FUNCTION_BLOCK IO_DI32 (* Cartao TM3DI32K da remota TM3BCEIP: separa as 2 words lidas em 32 bits e publica cada bit por symlink, com depurador *)
  (* Standard: 61499-2 *)
  (* Version 1.0, 10/2/2026, Hidryco, Hidryco, Baseado em TM_DI32/TM_DO32 e DI_TESTE; inclui gate de comunicacao *)
  PACKAGE Hidryco.HidrycoLib;
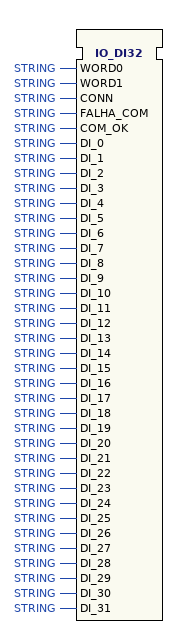
  VAR_INPUT
    WORD0 : STRING; (* Nome do symlink da word 0 do cartao (bits 0-15), ex.: A3_I0_0_15 *)
    WORD1 : STRING; (* Nome do symlink da word 1 do cartao (bits 16-31) *)
    CONN : STRING; (* Nome do symlink connStatusInt da remota, ex.: A2_REMOTA1_CONN_STATUS_INT (obrigatorio: sem ele o cartao fica em falha) *)
    FALHA_COM : STRING; (* Nome do symlink BOOL publicado com a falha de comunicacao do cartao (TRUE = remota offline) *)
    COM_OK : STRING; (* Nome do symlink BOOL publicado com comunicacao OK (TRUE = remota online) *)
    DI_0 : STRING; (* Nome do symlink BOOL publicado para o bit 0 do cartao *)
    DI_1 : STRING; (* Nome do symlink BOOL publicado para o bit 1 do cartao *)
    DI_2 : STRING; (* Nome do symlink BOOL publicado para o bit 2 do cartao *)
    DI_3 : STRING; (* Nome do symlink BOOL publicado para o bit 3 do cartao *)
    DI_4 : STRING; (* Nome do symlink BOOL publicado para o bit 4 do cartao *)
    DI_5 : STRING; (* Nome do symlink BOOL publicado para o bit 5 do cartao *)
    DI_6 : STRING; (* Nome do symlink BOOL publicado para o bit 6 do cartao *)
    DI_7 : STRING; (* Nome do symlink BOOL publicado para o bit 7 do cartao *)
    DI_8 : STRING; (* Nome do symlink BOOL publicado para o bit 8 do cartao *)
    DI_9 : STRING; (* Nome do symlink BOOL publicado para o bit 9 do cartao *)
    DI_10 : STRING; (* Nome do symlink BOOL publicado para o bit 10 do cartao *)
    DI_11 : STRING; (* Nome do symlink BOOL publicado para o bit 11 do cartao *)
    DI_12 : STRING; (* Nome do symlink BOOL publicado para o bit 12 do cartao *)
    DI_13 : STRING; (* Nome do symlink BOOL publicado para o bit 13 do cartao *)
    DI_14 : STRING; (* Nome do symlink BOOL publicado para o bit 14 do cartao *)
    DI_15 : STRING; (* Nome do symlink BOOL publicado para o bit 15 do cartao *)
    DI_16 : STRING; (* Nome do symlink BOOL publicado para o bit 16 do cartao *)
    DI_17 : STRING; (* Nome do symlink BOOL publicado para o bit 17 do cartao *)
    DI_18 : STRING; (* Nome do symlink BOOL publicado para o bit 18 do cartao *)
    DI_19 : STRING; (* Nome do symlink BOOL publicado para o bit 19 do cartao *)
    DI_20 : STRING; (* Nome do symlink BOOL publicado para o bit 20 do cartao *)
    DI_21 : STRING; (* Nome do symlink BOOL publicado para o bit 21 do cartao *)
    DI_22 : STRING; (* Nome do symlink BOOL publicado para o bit 22 do cartao *)
    DI_23 : STRING; (* Nome do symlink BOOL publicado para o bit 23 do cartao *)
    DI_24 : STRING; (* Nome do symlink BOOL publicado para o bit 24 do cartao *)
    DI_25 : STRING; (* Nome do symlink BOOL publicado para o bit 25 do cartao *)
    DI_26 : STRING; (* Nome do symlink BOOL publicado para o bit 26 do cartao *)
    DI_27 : STRING; (* Nome do symlink BOOL publicado para o bit 27 do cartao *)
    DI_28 : STRING; (* Nome do symlink BOOL publicado para o bit 28 do cartao *)
    DI_29 : STRING; (* Nome do symlink BOOL publicado para o bit 29 do cartao *)
    DI_30 : STRING; (* Nome do symlink BOOL publicado para o bit 30 do cartao *)
    DI_31 : STRING; (* Nome do symlink BOOL publicado para o bit 31 do cartao *)
  END_VAR
  FBS
    plcStart1 : plcStart(Prio := 3);
    IThis : IO_DI32_HMI(QI := TRUE);
    DST_CONN : SYMLINKMULTIVARDST_5A03F112CD5D470(QI := TRUE); {SET_ATTRIBUTE(Configuration.GenericFBType.InterfaceParams, Runtime.System#I:=1;VALUE${I$}:INT)}
    DST_W0 : SYMLINKMULTIVARDST_5A03F112CD5D470(QI := TRUE); {SET_ATTRIBUTE(Configuration.GenericFBType.InterfaceParams, Runtime.System#I:=1;VALUE${I$}:INT)}
    DST_W1 : SYMLINKMULTIVARDST_5A03F112CD5D470(QI := TRUE); {SET_ATTRIBUTE(Configuration.GenericFBType.InterfaceParams, Runtime.System#I:=1;VALUE${I$}:INT)}
    Gate : basicIOComGate;
    I2W_0 : ANY2ANY_100577755E31233DE; {SET_ATTRIBUTE(Configuration.GenericFBType.InterfaceParams, Runtime.Standard#CNT:=1;IN${CNT$}:INT;OUT${CNT$}:WORD)}
    SPLIT_0 : BITMAN_1879143E4E6E9A030; {SET_ATTRIBUTE(Configuration.GenericFBType.InterfaceParams, Runtime.Standard#CNTIN:=1;CNTOUT:=16;IN${CNTIN$}:WORD;OUT${CNTOUT$}:BOOL,BOOL,BOOL,BOOL,BOOL,BOOL,BOOL,BOOL,BOOL,BOOL,BOOL,BOOL,BOOL,BOOL,BOOL,BOOL)}
    SRC_B0 : SYMLINKMULTIVARSRC_854A896E88500D19(QI := TRUE); {SET_ATTRIBUTE(Configuration.GenericFBType.InterfaceParams, Runtime.System#I:=16;VALUE${I$}:BOOL,BOOL,BOOL,BOOL,BOOL,BOOL,BOOL,BOOL,BOOL,BOOL,BOOL,BOOL,BOOL,BOOL,BOOL,BOOL)}
    I2W_1 : ANY2ANY_100577755E31233DE; {SET_ATTRIBUTE(Configuration.GenericFBType.InterfaceParams, Runtime.Standard#CNT:=1;IN${CNT$}:INT;OUT${CNT$}:WORD)}
    SPLIT_1 : BITMAN_1879143E4E6E9A030; {SET_ATTRIBUTE(Configuration.GenericFBType.InterfaceParams, Runtime.Standard#CNTIN:=1;CNTOUT:=16;IN${CNTIN$}:WORD;OUT${CNTOUT$}:BOOL,BOOL,BOOL,BOOL,BOOL,BOOL,BOOL,BOOL,BOOL,BOOL,BOOL,BOOL,BOOL,BOOL,BOOL,BOOL)}
    SRC_B1 : SYMLINKMULTIVARSRC_854A896E88500D19(QI := TRUE); {SET_ATTRIBUTE(Configuration.GenericFBType.InterfaceParams, Runtime.System#I:=16;VALUE${I$}:BOOL,BOOL,BOOL,BOOL,BOOL,BOOL,BOOL,BOOL,BOOL,BOOL,BOOL,BOOL,BOOL,BOOL,BOOL,BOOL)}
    SRC_FALHA : SYMLINKMULTIVARSRC_277E97BEC1451D2C(QI := TRUE); {SET_ATTRIBUTE(Configuration.GenericFBType.InterfaceParams, Runtime.System#I:=2;VALUE${I$}:BOOL,BOOL)}
  END_FBS
  EVENT_CONNECTIONS
    DST_W0.CNF TO Gate.BD23A685891FD57E;
    DST_W1.CNF TO Gate.BD23A685891FD57E;
    DST_CONN.CNF TO Gate.BD23A685891FD57E;
    Gate.B07445CE7289017B TO I2W_0.REQ;
    I2W_0.CNF TO SPLIT_0.REQ;
    SPLIT_0.CNF TO SRC_B0.REQ;
    SPLIT_0.CNF TO IThis.48E8D870A969746E;
    Gate.B07445CE7289017B TO I2W_1.REQ;
    I2W_1.CNF TO SPLIT_1.REQ;
    SPLIT_1.CNF TO SRC_B1.REQ;
    SPLIT_1.CNF TO IThis.48E8D870A969746E;
    Gate.B07445CE7289017B TO SRC_FALHA.REQ;
    Gate.B07445CE7289017B TO IThis.48E8D870A969746E;
    plcStart1.FIRST_INIT TO DST_W0.INIT;
    plcStart1.REDO_INIT TO DST_W0.INIT;
    DST_W0.INITO TO DST_W1.INIT;
    DST_W1.INITO TO DST_CONN.INIT;
    DST_CONN.INITO TO SPLIT_0.INIT;
    SPLIT_0.INITO TO SPLIT_1.INIT;
    SPLIT_1.INITO TO SRC_B0.INIT;
    SRC_B0.INITO TO SRC_B1.INIT;
    SRC_B1.INITO TO SRC_FALHA.INIT;
    SRC_FALHA.INITO TO IThis.750DD2BDCC8DF380;
    IThis.57A7ED843B74E1C5 TO plcStart1.ACK_FIRST;
  END_CONNECTIONS
  DATA_CONNECTIONS
    DST_W0.VALUE1 TO Gate.E55C0654C443D12C;
    DST_W1.VALUE1 TO Gate.1DD6D86783AAC6A7;
    DST_CONN.VALUE1 TO Gate.802FC2CA3041A58B;
    Gate.46D4D28C21794752 TO I2W_0.IN1;
    I2W_0.OUT1 TO SPLIT_0.IN1;
    SPLIT_0.OUT1 TO SRC_B0.VALUE1;
    SPLIT_0.OUT1 TO IThis.C9873E75BAB2C979;
    DI_0 TO SRC_B0.NAME1;
    SPLIT_0.OUT2 TO SRC_B0.VALUE2;
    SPLIT_0.OUT2 TO IThis.54DAA12BA959314B;
    DI_1 TO SRC_B0.NAME2;
    SPLIT_0.OUT3 TO SRC_B0.VALUE3;
    SPLIT_0.OUT3 TO IThis.A0F1798486889AB9;
    DI_2 TO SRC_B0.NAME3;
    SPLIT_0.OUT4 TO SRC_B0.VALUE4;
    SPLIT_0.OUT4 TO IThis.DAB6BF4E12DE60FB;
    DI_3 TO SRC_B0.NAME4;
    SPLIT_0.OUT5 TO SRC_B0.VALUE5;
    SPLIT_0.OUT5 TO IThis.B5AE01A427636046;
    DI_4 TO SRC_B0.NAME5;
    SPLIT_0.OUT6 TO SRC_B0.VALUE6;
    SPLIT_0.OUT6 TO IThis.51B49F6913B79E94;
    DI_5 TO SRC_B0.NAME6;
    SPLIT_0.OUT7 TO SRC_B0.VALUE7;
    SPLIT_0.OUT7 TO IThis.085D597396FFF72B;
    DI_6 TO SRC_B0.NAME7;
    SPLIT_0.OUT8 TO SRC_B0.VALUE8;
    SPLIT_0.OUT8 TO IThis.6CE6A2F9B1A36CA8;
    DI_7 TO SRC_B0.NAME8;
    SPLIT_0.OUT9 TO SRC_B0.VALUE9;
    SPLIT_0.OUT9 TO IThis.77FA22E1E5901DF6;
    DI_8 TO SRC_B0.NAME9;
    SPLIT_0.OUT10 TO SRC_B0.VALUE10;
    SPLIT_0.OUT10 TO IThis.35713C99BB0D6DF9;
    DI_9 TO SRC_B0.NAME10;
    SPLIT_0.OUT11 TO SRC_B0.VALUE11;
    SPLIT_0.OUT11 TO IThis.B7CDDE68FB84038A;
    DI_10 TO SRC_B0.NAME11;
    SPLIT_0.OUT12 TO SRC_B0.VALUE12;
    SPLIT_0.OUT12 TO IThis.EE477D3BD3D6005B;
    DI_11 TO SRC_B0.NAME12;
    SPLIT_0.OUT13 TO SRC_B0.VALUE13;
    SPLIT_0.OUT13 TO IThis.FD676144D2357993;
    DI_12 TO SRC_B0.NAME13;
    SPLIT_0.OUT14 TO SRC_B0.VALUE14;
    SPLIT_0.OUT14 TO IThis.1152BF33A398D083;
    DI_13 TO SRC_B0.NAME14;
    SPLIT_0.OUT15 TO SRC_B0.VALUE15;
    SPLIT_0.OUT15 TO IThis.9637F813B8B3D403;
    DI_14 TO SRC_B0.NAME15;
    SPLIT_0.OUT16 TO SRC_B0.VALUE16;
    SPLIT_0.OUT16 TO IThis.B365DC456E4012C2;
    DI_15 TO SRC_B0.NAME16;
    Gate.42FBD7F29792C6AD TO I2W_1.IN1;
    I2W_1.OUT1 TO SPLIT_1.IN1;
    SPLIT_1.OUT1 TO SRC_B1.VALUE1;
    SPLIT_1.OUT1 TO IThis.136C56BFB7CFC592;
    DI_16 TO SRC_B1.NAME1;
    SPLIT_1.OUT2 TO SRC_B1.VALUE2;
    SPLIT_1.OUT2 TO IThis.794300F27541D1C3;
    DI_17 TO SRC_B1.NAME2;
    SPLIT_1.OUT3 TO SRC_B1.VALUE3;
    SPLIT_1.OUT3 TO IThis.B15F030F6C285371;
    DI_18 TO SRC_B1.NAME3;
    SPLIT_1.OUT4 TO SRC_B1.VALUE4;
    SPLIT_1.OUT4 TO IThis.D864A0B80A091C75;
    DI_19 TO SRC_B1.NAME4;
    SPLIT_1.OUT5 TO SRC_B1.VALUE5;
    SPLIT_1.OUT5 TO IThis.A5AFCC991D7A6F52;
    DI_20 TO SRC_B1.NAME5;
    SPLIT_1.OUT6 TO SRC_B1.VALUE6;
    SPLIT_1.OUT6 TO IThis.DA9AB5F1447847F6;
    DI_21 TO SRC_B1.NAME6;
    SPLIT_1.OUT7 TO SRC_B1.VALUE7;
    SPLIT_1.OUT7 TO IThis.FA441CBAF33D6A91;
    DI_22 TO SRC_B1.NAME7;
    SPLIT_1.OUT8 TO SRC_B1.VALUE8;
    SPLIT_1.OUT8 TO IThis.7D78689BD8D3A131;
    DI_23 TO SRC_B1.NAME8;
    SPLIT_1.OUT9 TO SRC_B1.VALUE9;
    SPLIT_1.OUT9 TO IThis.3CD56822DF3156FF;
    DI_24 TO SRC_B1.NAME9;
    SPLIT_1.OUT10 TO SRC_B1.VALUE10;
    SPLIT_1.OUT10 TO IThis.378E886E7460846B;
    DI_25 TO SRC_B1.NAME10;
    SPLIT_1.OUT11 TO SRC_B1.VALUE11;
    SPLIT_1.OUT11 TO IThis.228786A835508E0D;
    DI_26 TO SRC_B1.NAME11;
    SPLIT_1.OUT12 TO SRC_B1.VALUE12;
    SPLIT_1.OUT12 TO IThis.E509173F2903142D;
    DI_27 TO SRC_B1.NAME12;
    SPLIT_1.OUT13 TO SRC_B1.VALUE13;
    SPLIT_1.OUT13 TO IThis.6DE9A756559B31D8;
    DI_28 TO SRC_B1.NAME13;
    SPLIT_1.OUT14 TO SRC_B1.VALUE14;
    SPLIT_1.OUT14 TO IThis.5E6CEA4A9BFAA536;
    DI_29 TO SRC_B1.NAME14;
    SPLIT_1.OUT15 TO SRC_B1.VALUE15;
    SPLIT_1.OUT15 TO IThis.2988D15A72D1D754;
    DI_30 TO SRC_B1.NAME15;
    SPLIT_1.OUT16 TO SRC_B1.VALUE16;
    SPLIT_1.OUT16 TO IThis.D9A2D37279245CA5;
    DI_31 TO SRC_B1.NAME16;
    Gate.67074C7AC6CF1B2E TO SRC_FALHA.VALUE1;
    Gate.E7CF4253A5649388 TO SRC_FALHA.VALUE2;
    FALHA_COM TO SRC_FALHA.NAME1;
    COM_OK TO SRC_FALHA.NAME2;
    WORD0 TO DST_W0.NAME1;
    WORD1 TO DST_W1.NAME1;
    CONN TO DST_CONN.NAME1;
    Gate.67074C7AC6CF1B2E TO IThis.50A5B3E4E7FDBBC6;
    DST_W0.VALUE1 TO IThis.3EC5D9E54559DB42;
    DST_W1.VALUE1 TO IThis.9F3EA8F732D0F44D;
    DST_CONN.VALUE1 TO IThis.1E240E86070AE622;
  END_CONNECTIONS
END_FUNCTION_BLOCK
